FUNCTION_BLOCK FB_MoverApplication IMPLEMENTS I_MoverApplication
VAR
	ipMoverStandard	: I_XPlanarMoverStandard;
	fbMoverStandard	: FB_XPlanarMoverStandard;

	
	nMoverIndex		: INT;
	
	nTrackId		: UDINT;
	
	// customer Data
	bIsLoaded		: BOOL;	
		
		
	// customer templates
	fbSwivelMovement 	: FB_SwivelMovement;
	ipSwivelMovement	: I_SwivelMovement;	
	
	fbShakeMovement 	: FB_ShakeMovement;
	ipShakeMovement		: I_ShakeMovement;		
	
	fbGCode			: FB_GCode;
	ipGCode			: I_GCode;
	
	
		
END_VAR

VAR_OUTPUT
	VisuPos	: MoverVector;
END_VAR

METHOD Cycle
ipMoverStandard := fbMoverStandard;


IF std <> 0 THEN
	std.cycle();
	VisuPos := std.P_ActPosition;
END_IF



// additional functionality
ipSwivelMovement := fbSwivelMovement;
fbSwivelMovement(ipMover := ipMoverStandard);
fbSwivelMovement.Cycle();


ipShakeMovement := fbShakeMovement;
fbShakeMovement(ipMover := ipMoverStandard);
fbShakeMovement.Cycle();

ipGCode := fbGCode;
fbGCode(ipMover := ipMoverStandard);
fbGCode.Cycle();
END_METHOD

PROPERTY GCode : I_GCode
GET
IF ipGCode <> 0 THEN
	GCode := ipGCode;	
END_IF
END_GET
SET
ipGCode := GCode;
END_SET
END_PROPERTY

PROPERTY P_nMoverIndex : INT
GET
P_nMoverIndex := nMoverIndex;
END_GET
SET
nMoverIndex := P_nMoverIndex;
END_SET
END_PROPERTY

PROPERTY P_nTrackId : UDINT
GET
P_nTrackId := nTrackId;
END_GET
SET
nTrackId := P_nTrackId;
END_SET
END_PROPERTY

PROPERTY Shake : I_ShakeMovement
GET
IF ipShakeMovement <> 0 THEN
	Shake := ipShakeMovement;	
END_IF
END_GET
SET
ipShakeMovement := Shake;
END_SET
END_PROPERTY

PROPERTY std : I_XPlanarMoverStandard
GET
IF ipMoverStandard <> 0 THEN
	std := ipMoverStandard;	
END_IF
END_GET
SET
ipMoverStandard := std;
END_SET
END_PROPERTY

PROPERTY Swivel : I_SwivelMovement
GET
IF ipSwivelMovement <> 0 THEN
	Swivel := ipSwivelMovement;	
END_IF
END_GET
SET
ipSwivelMovement := Swivel;
END_SET
END_PROPERTY

END_FUNCTION_BLOCK

(* stored: Version 1.1.0.1
   POU FB_MoverApplication: Id {c04d6286-3029-4c56-b1dc-fb0bc59440b4}, SpecialFunc None
   Method Cycle: Id {3cff7639-35c1-4bdb-9020-86adc6f8ac20}
   Property GCode: Id {d6ceba06-f2f9-44b5-9e9b-5229362f963b}
   Get Get: Id {53cfb764-9642-455a-9b1a-e61988470247}
   Set Set: Id {01c10ac2-7699-494a-b7c9-da151e5a620a}
   Property P_nMoverIndex: Id {24fd9882-3bd1-494e-af6d-7436ababb6c7}
   Get Get: Id {7e7ff66a-0a50-4673-a237-4c68a9caf0f1}
   Set Set: Id {8dc969a4-7930-4648-8576-11abf341d667}
   Property P_nTrackId: Id {1adb6d69-ee83-4794-991d-ba156490540f}
   Get Get: Id {6474aff8-cc6e-4030-a00d-3795177ba84b}
   Set Set: Id {afc56916-c8fa-48e5-b821-a8c829d72231}
   Property Shake: Id {fe7a1c72-c8ee-4fc3-93c8-86afb91fcc60}
   Get Get: Id {bd0efa6c-6a08-4fa6-95ec-316dd8e03661}
   Set Set: Id {612209d5-e739-4406-9176-b00d4b63d651}
   Property std: Id {87d8a23e-7c73-4ac0-b107-cdf4f71a1360}
   Get Get: Id {7d6b3eb7-03c1-44d4-b5d7-de62390f59c9}
   Set Set: Id {b6ec7cab-1d1c-4ee6-8861-a1dcde7e9843}
   Property Swivel: Id {15aaee38-ef1c-4b1e-a501-c916248227d1}
   Get Get: Id {734e2dc6-6f4e-4f12-af83-40aa87807527}
   Set Set: Id {58838ad0-be68-4044-b5c5-ca0997df969b} *)
